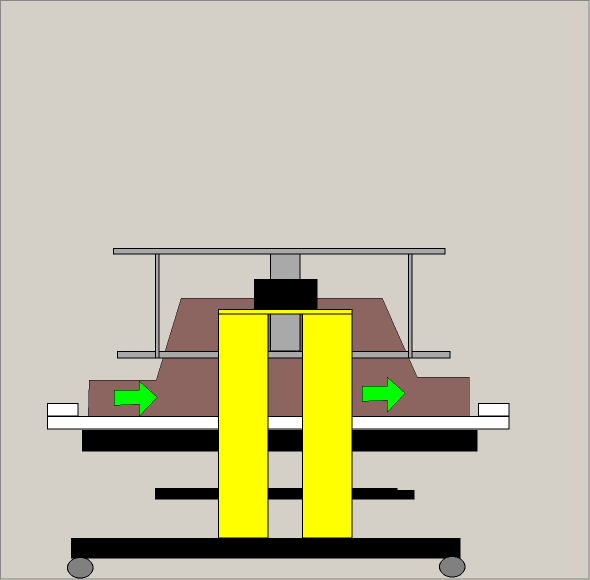
VISUALIZATION loadSpaScreen  // 590x580
    Rectangle (47,416 462x13)
    Polygon (88,416) (89,380) (156,380) (181,298) (382,298) (417,377) (469,377) (469,415) (469,416)
    Rectangle (236,287 98x30), angle 90
    Rectangle (117,351 333x7)
    Rectangle (155,488 242x11), angle 25
    Rectangle (171,490 243x9), angle 336
    Rectangle (82,430 395x21)
    Rectangle (71,538 389x20)
    Rectangle (218,313 50x225)
    Rectangle (302,313 50x225)
    Ellipse (439,556 26x21)
    Ellipse (67,557 26x21)
    Rectangle (218,309 134x5)
    Rectangle (254,279 63x30)
    Rectangle (408,253 4x105)
    Rectangle (155,253 4x105)
    Rectangle (113,248 332x6)
    Polygon (114,400) (114,405) (139,404) (139,416) (157,397) (139,381) (139,390) (114,390)
    Polygon (362,396) (362,401) (387,400) (387,412) (405,393) (387,377) (387,386) (362,386)
    Rectangle (478,403 31x13)
    Rectangle (47,403 31x13)
END_VISUALIZATION

(* stored: Version 1.1.0.1, ProductVersion 3.1.4024.15
   Visu loadSpaScreen: Id {fe1fb8c4-75aa-4d5c-9e19-9f2fa226d97c} *)
